Fanuc KAREL source: GET_POS_TYP.kl

PROGRAM T
%NOLOCKGROUP
VAR
 v0 : INTEGER
 v1 : INTEGER
 v2 : INTEGER
 v3 : INTEGER
 v4 : INTEGER
 v5 : INTEGER
BEGIN
 GET_POS_TYP(v0, v1, v2, v3, v4, v5)
END T
